{attribute 'obsolete' := 'Use E_EpicsInOut'}
TYPE ENUM_EpicsInOut : E_EpicsInOut; END_TYPE

(* stored: Version 1.1.0.1
   DUT ENUM_EpicsInOut: Id {eb849dbe-cc3c-4665-84db-6a2eb274e6d2} *)
